FUNCTION_BLOCK AbfolgeC (* Abfolge als Composite *)
  (* Standard: 61499-2 *)
  (* Version 1.0, 2022-10-10, franz *)
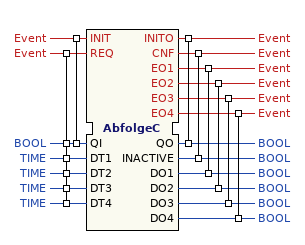
  EVENT_INPUT
    INIT WITH QI; (* Initialization Request *)
    REQ WITH QI, DT1, DT2, DT3, DT4; (* Normal Execution Request *)
  END_EVENT
  EVENT_OUTPUT
    INITO WITH QO; (* Initialization Confirm *)
    CNF WITH INACTIVE;
    EO1 WITH DO1;
    EO2 WITH DO2;
    EO3 WITH DO3;
    EO4 WITH DO4;
  END_EVENT
  VAR_INPUT
    QI : BOOL; (* Input event qualifier *)
    DT1 : TIME;
    DT2 : TIME;
    DT3 : TIME;
    DT4 : TIME;
  END_VAR
  VAR_OUTPUT
    QO : BOOL; (* Output event qualifier *)
    INACTIVE : BOOL;
    DO1 : BOOL;
    DO2 : BOOL;
    DO3 : BOOL;
    DO4 : BOOL;
  END_VAR
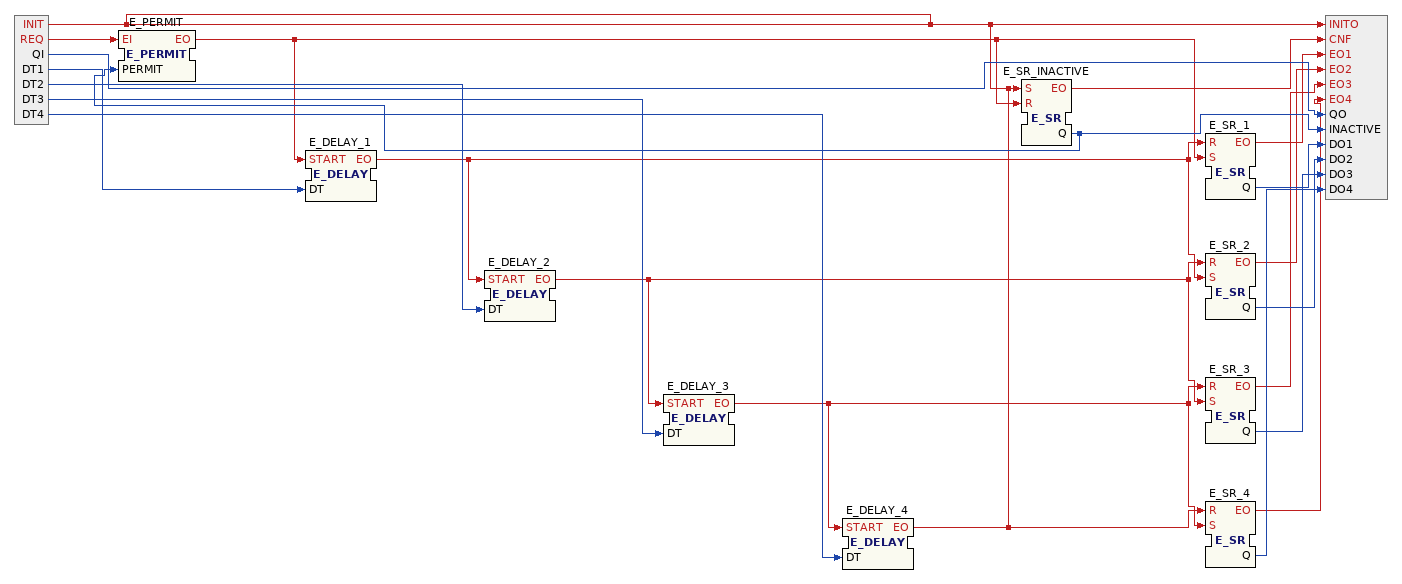
  FBS
    E_DELAY_1 : E_DELAY;
    E_DELAY_2 : E_DELAY;
    E_DELAY_3 : E_DELAY;
    E_DELAY_4 : E_DELAY;
    E_SR_1 : E_SR;
    E_SR_2 : E_SR;
    E_SR_3 : E_SR;
    E_SR_4 : E_SR;
    E_SR_INACTIVE : E_SR;
    E_PERMIT : E_PERMIT;
  END_FBS
  EVENT_CONNECTIONS
    E_DELAY_1.EO TO E_SR_1.R;
    E_DELAY_2.EO TO E_SR_2.R;
    E_DELAY_3.EO TO E_SR_3.R;
    E_DELAY_4.EO TO E_SR_4.R;
    E_DELAY_1.EO TO E_SR_2.S;
    E_DELAY_2.EO TO E_SR_3.S;
    E_DELAY_3.EO TO E_SR_4.S;
    E_DELAY_1.EO TO E_DELAY_2.START;
    E_DELAY_2.EO TO E_DELAY_3.START;
    E_DELAY_3.EO TO E_DELAY_4.START;
    INIT TO INITO;
    E_SR_1.EO TO EO1;
    E_SR_2.EO TO EO2;
    E_SR_3.EO TO EO3;
    E_SR_4.EO TO EO4;
    E_PERMIT.EO TO E_SR_1.S;
    E_PERMIT.EO TO E_DELAY_1.START;
    REQ TO E_PERMIT.EI;
    INIT TO E_SR_INACTIVE.S;
    E_DELAY_4.EO TO E_SR_INACTIVE.S;
    E_PERMIT.EO TO E_SR_INACTIVE.R;
    E_SR_INACTIVE.EO TO CNF;
  END_CONNECTIONS
  DATA_CONNECTIONS
    E_SR_1.Q TO DO1;
    E_SR_2.Q TO DO2;
    E_SR_3.Q TO DO3;
    E_SR_4.Q TO DO4;
    DT4 TO E_DELAY_4.DT;
    DT3 TO E_DELAY_3.DT;
    DT2 TO E_DELAY_2.DT;
    DT1 TO E_DELAY_1.DT;
    QI TO QO;
    E_SR_INACTIVE.Q TO INACTIVE;
    E_SR_INACTIVE.Q TO E_PERMIT.PERMIT;
  END_CONNECTIONS
END_FUNCTION_BLOCK
